KUKA KRL program: f_fraes2.src, f_fraes2.dat

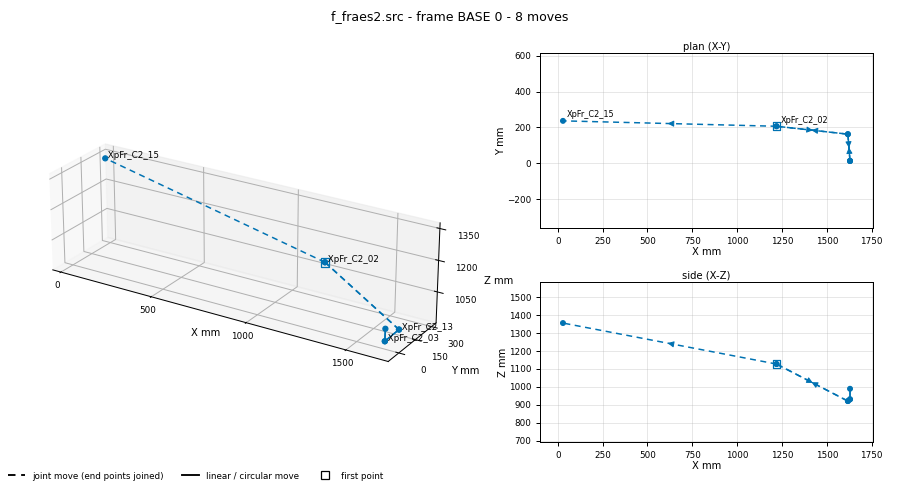
[picture p0: tool path of f_fraes2.src in frame BASE 0, 8 of 9 moves have a stored position in this frame; points joined in program order, loops and branches not executed]
--- f_fraes2.src ---
&ACCESS RVO3
&REL 37
&COMMENT Fresa C2
&PARAM DISKPATH = KRC:\R1\Program\SERVICE
&PARAM TEMPLATE = C:\KRC\Roboter\Template\vorgabe
&PARAM EDITMASK = *
DEF F_fraes2( )
;FOLD INI
  ;FOLD BASISTECH INI
    GLOBAL INTERRUPT DECL 3 WHEN $STOPMESS==TRUE DO IR_STOPM ( )
    INTERRUPT ON 3
    BAS (#INITMOV,0 )
  ;ENDFOLD (BASISTECH INI)
;FOLD SPOTTECH INI
USERSPOT(#INIT)
;ENDFOLD (SPOTTECH INI)
;FOLD GRIPPERTECH INI
USER_GRP(0,DUMMY,DUMMY,GDEFAULT)
;ENDFOLD (GRIPPERTECH INI)
  ;FOLD USER INI
    ;Make your modifications here

  ;ENDFOLD (USER INI)
;ENDFOLD (INI)

; Caracterização dos meios de produção:
; Versão Atual:
; 15/07/2013 12:00 Name: P13.050-R4 CHANGES: Fresa
; C2


chk_w2_wechs_ok ( )     ; CHECK FERRAMENTA: C2


;FOLD PTP Prf CONT Vel=100 % PDAT13 Tool[2]:GUN C2 Base[2]:ACCELO;%{PE}%R 8.2.20,%MKUKATPBASIS,%CMOVE,%VPTP,%P 1:PTP, 2:Prf, 3:C_DIS, 5:100, 7:PDAT13
$BWDSTART=FALSE
PDAT_ACT=PPDAT13
FDAT_ACT=FPrf
BAS(#PTP_PARAMS,100)
PTP XPrf C_DIS
;ENDFOLD
;FOLD PTP pFr_C2_02 CONT Vel=100 % PDAT2 Tool[2]:GUN C2 Base[2]:ACCELO;%{PE}%R 8.2.20,%MKUKATPBASIS,%CMOVE,%VPTP,%P 1:PTP, 2:pFr_C2_02, 3:C_DIS, 5:100, 7:PDAT2
$BWDSTART=FALSE
PDAT_ACT=PPDAT2
FDAT_ACT=FpFr_C2_02
BAS(#PTP_PARAMS,100)
PTP XpFr_C2_02 C_DIS
;ENDFOLD
;FOLD PTP pFr_C2_13 CONT Vel=100 % PDAT0 Tool[2]:GUN C2 Base[2]:ACCELO;%{PE}%R 8.2.20,%MKUKATPBASIS,%CMOVE,%VPTP,%P 1:PTP, 2:pFr_C2_13, 3:C_DIS, 5:100, 7:PDAT0
$BWDSTART=FALSE
PDAT_ACT=PPDAT0
FDAT_ACT=FpFr_C2_13
BAS(#PTP_PARAMS,100)
PTP XpFr_C2_13 C_DIS
;ENDFOLD

;FOLD LIN pFr_C2_03 CONT Vel=1 m/s CPDAT1 Tool[2]:GUN C2 Base[2]:ACCELO;%{PE}%R 8.2.20,%MKUKATPBASIS,%CMOVE,%VLIN,%P 1:LIN, 2:pFr_C2_03, 3:C_DIS C_DIS, 5:1, 7:CPDAT1
$BWDSTART=FALSE
LDAT_ACT=LCPDAT1
FDAT_ACT=FpFr_C2_03
BAS(#CP_PARAMS,1)
LIN XpFr_C2_03 C_DIS C_DIS
;ENDFOLD

;FOLD ; PONTO DE FRESAGEM;%{PE}%R 8.2.20,%MKUKATPBASIS,%CCOMMENT,%VNORMAL,%P 2:PONTO  DE  FRESAGEM
;ENDFOLD
;FOLD TIP.LIN_ Dress_01, Spot Gun 2 , RETR open , Tool[2], Base[0], EXT.TCP=FALSE;%{PE}%MKUKATPUSER
FDAT_ACT=FDress_01
BAS(#FRAMES)
LIN  XDress_01
S_ACT.GUN=2
S_ACT.RETR=#opn
S_READY=FALSE
USERSPOT (#DRESS,S_ACT )
WAIT FOR  S_READY
;ENDFOLD

;FOLD LIN pFr_C2_05 Vel=1 m/s CPDAT3 Tool[2]:GUN C2 Base[0];%{PE}%R 8.2.20,%MKUKATPBASIS,%CMOVE,%VLIN,%P 1:LIN, 2:pFr_C2_05, 3:, 5:1, 7:CPDAT3
$BWDSTART=FALSE
LDAT_ACT=LCPDAT3
FDAT_ACT=FpFr_C2_05
BAS(#CP_PARAMS,1)
LIN XpFr_C2_05
;ENDFOLD

;FOLD PTP pFr_C2_10 PDAT6 SPOT Gun=2 RETR OPN PgNo1=125 ACTIVE=1 Tool[2]:GUN C2 Base[0];%{PE}%R 8.2.2,%MKUKATPSPOT,%CSPOT,%VPTP,%P 1:PTP, 2:pFr_C2_10, 3:, 5:100, 7:PDAT6, 10:2, 12:#FIRST, 14:#OPN, 16:125, 18:1, 20:0, 22:0, 24:1, 25:NORMAL
$BWDSTART=FALSE
PDAT_ACT=PPDAT6
FDAT_ACT=FpFr_C2_10
BAS(#PTP_PARAMS,PPDAT6.VEL)
S_ACT.GUN=2
S_ACT.PAIR=SDEFAULT.PAIR
S_ACT.RETR=#OPN
S_ACT.CLO_TM=1
S_ACT.PGNO1=125
S_ACT.PGNO2=SDEFAULT.PGNO2
S_ACT.PRESS1=SDEFAULT.PRESS1
S_ACT.PRESS2=SDEFAULT.PRESS2
S_READY=FALSE
PTP XpFr_C2_10
USERSPOT(#SPOT, S_ACT)
WAIT FOR S_READY
;ENDFOLD
;FOLD PTP pFr_C2_07 CONT Vel=100 % PDAT4 Tool[2]:GUN C2 Base[2]:ACCELO;%{PE}%R 8.2.20,%MKUKATPBASIS,%CMOVE,%VPTP,%P 1:PTP, 2:pFr_C2_07, 3:C_DIS, 5:100, 7:PDAT4
$BWDSTART=FALSE
PDAT_ACT=PPDAT4
FDAT_ACT=FpFr_C2_07
BAS(#PTP_PARAMS,100)
PTP XpFr_C2_07 C_DIS
;ENDFOLD
;FOLD PTP pFr_C2_15 CONT Vel=100 % PDAT12 Tool[2]:GUN C2 Base[2]:ACCELO;%{PE}%R 8.2.20,%MKUKATPBASIS,%CMOVE,%VPTP,%P 1:PTP, 2:pFr_C2_15, 3:C_DIS, 5:100, 7:PDAT12
$BWDSTART=FALSE
PDAT_ACT=PPDAT12
FDAT_ACT=FpFr_C2_15
BAS(#PTP_PARAMS,100)
PTP XpFr_C2_15 C_DIS
;ENDFOLD




END

--- f_fraes2.dat ---
&ACCESS RVO3
&REL 37
&COMMENT Fresa C2
&PARAM DISKPATH = KRC:\R1\Program\SERVICE
&PARAM TEMPLATE = C:\KRC\Roboter\Template\vorgabe
&PARAM EDITMASK = *
DEFDAT  f_fraes2
;FOLD EXTERNAL DECLARATIONS;%{PE}%MKUKATPBASIS,%CEXT,%VCOMMON,%P
;FOLD GRIPPERTECH EXT
EXT  H50 (INT  :IN,INT  :IN,INT  :IN,GRP_TYP  :IN )
;ENDFOLD (GRIPPERTECH EXT)
;FOLD SPOTTECH EXT
EXT  USERSPOT (S_COMMAND  :IN,SPOT_TYPE  :IN )
;ENDFOLD (SPOTTECH EXT)
;FOLD BASISTECH EXT;%{PE}%MKUKATPBASIS,%CEXT,%VEXT,%P
EXT  BAS (BAS_COMMAND  :IN,REAL  :IN )
DECL INT SUCCESS
;ENDFOLD (BASISTECH EXT)
;FOLD USER EXT;%{E}%MKUKATPUSER,%CEXT,%VEXT,%P
;Make your modifications here

;ENDFOLD (USER EXT)
;ENDFOLD (EXTERNAL DECLARATIONS)
DECL BASIS_SUGG_T LAST_BASIS={POINT1[] "P3                      ",POINT2[] "P3                      ",CP_PARAMS[] "CPDAT0                  ",PTP_PARAMS[] "PDAT15                  ",CONT[] "                        ",CP_VEL[] "2.0                     ",PTP_VEL[] "100                     ",SPL_NAME[] "S0                      "}
DECL PDAT PPDAT1={VEL 100.0,ACC 100.0,APO_DIST 100.0,APO_MODE #CDIS}
DECL E6POS XpFr_C2_01={X 629.392517,Y -514.732727,Z 1173.64001,A 141.479202,B 1.02019298,C 5.9837079,S 2,T 2,E1 -357.531708,E2 0.0,E3 0.0,E4 0.0,E5 0.0,E6 0.0}
DECL FDAT FpFr_C2_01={TOOL_NO 2,BASE_NO 0,IPO_FRAME #BASE,POINT2[] " ",TQ_STATE FALSE}
DECL E6POS XPFR_C2_02={X 1219.52002,Y 206.387299,Z 1127.48401,A -83.8557816,B -5.2056489,C -1.69778001,S 2,T 3,E1 -357.533112,E2 0.0,E3 0.0,E4 0.0,E5 0.0,E6 0.0}
DECL FDAT FpFr_C2_02={TOOL_NO 2,BASE_NO 0,IPO_FRAME #BASE,POINT2[] " ",TQ_STATE FALSE}
DECL PDAT PPDAT2={VEL 100.0,ACC 100.0,APO_DIST 100.0,APO_MODE #CDIS}
DECL E6POS XPFR_C2_03={X 1629.12097,Y 12.6184902,Z 930.869812,A -86.0264206,B -2.32755995,C -0.372054309,S 2,T 3,E1 -357.522186,E2 0.0,E3 0.0,E4 0.0,E5 0.0,E6 0.0}
DECL FDAT FpFr_C2_03={TOOL_NO 2,BASE_NO 0,IPO_FRAME #BASE,POINT2[] " ",TQ_STATE FALSE}
DECL LDAT LCPDAT1={VEL 2.0,ACC 100.0,APO_DIST 100.0,APO_FAC 50.0,AXIS_VEL 100.0,AXIS_ACC 100.0,ORI_TYP #VAR,CIRC_TYP #BASE,JERK_FAC 50.0,GEAR_JERK 50.0,EXAX_IGN 0}
DECL E6POS XPFR_C2_05={X 1629.12097,Y 12.6183004,Z 930.869995,A -86.0264282,B -2.32756209,C -0.37204501,S 2,T 3,E1 -357.522186,E2 0.0,E3 0.0,E4 0.0,E5 0.0,E6 0.0}
DECL FDAT FpFr_C2_05={TOOL_NO 2,BASE_NO 0,IPO_FRAME #BASE,POINT2[] " ",TQ_STATE FALSE}
DECL LDAT LCPDAT3={VEL 2.0,ACC 100.0,APO_DIST 100.0,APO_FAC 50.0,AXIS_VEL 100.0,AXIS_ACC 100.0,ORI_TYP #VAR,CIRC_TYP #BASE,JERK_FAC 50.0,GEAR_JERK 50.0,EXAX_IGN 0}
DECL E6POS XPFR_C2_07={X 1219.52002,Y 206.393707,Z 1127.48303,A -83.8551788,B -5.20540094,C -1.697837,S 2,T 3,E1 -357.533112,E2 0.0,E3 0.0,E4 0.0,E5 0.0,E6 0.0}
DECL FDAT FpFr_C2_07={TOOL_NO 2,BASE_NO 0,IPO_FRAME #BASE,POINT2[] " ",TQ_STATE FALSE}
DECL PDAT PPDAT4={VEL 100.0,ACC 100.0,APO_DIST 100.0,APO_MODE #CDIS}
DECL FDAT FDress_01={TOOL_NO 2,BASE_NO 0,IPO_FRAME #BASE}
DECL E6POS XDress_01={X 1629.30701,Y 14.0126696,Z 989.718323,A -91.6897736,B 0.0766007826,C -0.140863299,S 2,T 11,E1 -357.519196,E2 0.0,E3 0.0,E4 0.0,E5 0.0,E6 0.0}
DECL SPOT_SUGG_T LAST_SPOT={GUN[] "2                       ",RETR_CMD[] "#OPN                    ",CHOISE[] "#FIRST                  ",CLO_TM[] "1                       ",PGNO1[] "1                       ",PRESS1[] "0                       ",PGNO2[] "1                       ",PRESS2[] "0                       ",SPOT_PARAMS[] "NORMAL                  "}
DECL E6POS XPFR_C2_10={X 1617.37903,Y 162.361206,Z 920.988525,A -84.7256699,B -5.22538614,C -0.75706929,S 2,T 3,E1 -357.533112,E2 0.0,E3 0.0,E4 0.0,E5 0.0,E6 0.0}
DECL FDAT FpFr_C2_10={TOOL_NO 2,BASE_NO 0,IPO_FRAME #BASE,POINT2[] " ",TQ_STATE FALSE}
DECL PDAT PPDAT6={VEL 100.0,ACC 100.0,APO_DIST 100.0}
DECL PDAT PPDAT0={VEL 100.0,ACC 100.0,APO_DIST 100.0,APO_MODE #CDIS}
DECL E6POS XpFr_C2_13={X 1617.37695,Y 162.362106,Z 920.987976,A -84.7255173,B -5.22530985,C -0.75712502,S 2,T 3,E1 -357.533997,E2 0.0,E3 0.0,E4 0.0,E5 0.0,E6 0.0}
DECL FDAT FpFr_C2_13={TOOL_NO 2,BASE_NO 0,IPO_FRAME #BASE,POINT2[] " ",TQ_STATE FALSE}
DECL PDAT PPDAT11={VEL 100.0,ACC 100.0,APO_DIST 100.0,APO_MODE #CDIS}
DECL E6POS XpFr_C2_14={X 629.385071,Y -514.736816,Z 1173.64001,A 141.479095,B 1.02008903,C 5.98404408,S 2,T 2,E1 -357.531586,E2 0.0,E3 0.0,E4 0.0,E5 0.0,E6 0.0}
DECL FDAT FpFr_C2_14={TOOL_NO 2,BASE_NO 0,IPO_FRAME #BASE,POINT2[] " ",TQ_STATE FALSE}
DECL PDAT PPDAT12={VEL 100.0,ACC 100.0,APO_DIST 100.0,APO_MODE #CDIS}
DECL E6POS XpFr_C2_15={X 28.8758202,Y 236.546707,Z 1356.04297,A -94.0205002,B 5.74972391,C -0.112636402,S 2,T 3,E1 855.296692,E2 0.0,E3 0.0,E4 0.0,E5 0.0,E6 0.0}
DECL FDAT FpFr_C2_15={TOOL_NO 2,BASE_NO 0,IPO_FRAME #BASE,POINT2[] " ",TQ_STATE FALSE}
DECL PDAT PPDAT13={VEL 100.0,ACC 100.0,APO_DIST 100.0,APO_MODE #CDIS}
DECL E6POS XPrf={X -6773.34717,Y 2749.37598,Z -287.186707,A -4.02050114,B 5.74972391,C -0.112636402,S 2,T 3,E1 855.296692,E2 0.0,E3 0.0,E4 0.0,E5 0.0,E6 0.0}
DECL FDAT FPrf={TOOL_NO 2,BASE_NO 2,IPO_FRAME #BASE,POINT2[] " ",TQ_STATE FALSE}
ENDDAT
